FUNCTION alg_a: LREAL
VAR_INPUT
    state: STATE;
END_VAR


        alg_a := (state.cvar_c) + (derivcvar_c(state));

END_FUNCTION

(* stored: ProductVersion 3.1.0.18, Version 1.1.0.1 *)
